(* IEC 61131-3 sources: std_i2980_v2.06_cp053/Source/IMM/ieccontrol/GlobalBaseArchives (part 10) *)

(* ---- ABLintabLoader.pu ---- *)
(*
@h    ! WARNING !
@h    The Kemro K2 system (including software) only meets category B according to EN 954-1,
@h    thus it is not intended for usage in safety-relevant control applications in the field
@h    of personal safety (e.g. emergency stop).
@h    To implement potentially necessary safety-relevant control tasks, always use additional
@h    external safety devices that are intended for the particular purpose, and meet the necessary
@h    functional safety.
@h    For further information see EN 954-1 (EN ISO 13849-1) and/or the K2-x00 user manual, chapter
@h    "CE conformity, directives and standards".

lintab loader

@FunctionID: CR_0030048

*)

IMPORT_OVER_LISTFILE
 GET_RUNTIME
, KFILE_Open
, KFILE_Read
, KFILE_Close
, STRING_TO_ASCII
, KFILE_GetFirst
, KFILE_GetNext
, KCAT_GetHandle
, KCAT_GetValue
, CMD_LINTABLOAD
, CMD_LINTABLISTFILES
, cLTBLDR_ERR_UNKNOWNCMD
, KFILE_Mode_ReadOnly
, KFILE_Status_OK
, cLTBLDR_ERR_FILENOTFOUND
, cLTBLDR_ERR_OUTOFBOUND
, cLTBLDR_MAXFILES
, cLTBLDR_ERR_MAXFILESREACHED
, KCAT_Status_OK
, cLTBLDR_ROOTPATH
, tsLintabLoaderData
, KFILE_Status
, tsTraceLevel
, KFILE_Open_Data
, KCTRL_Lintab_Point
, KAPPL_LintabData
, KCAT_Status
, KCAT_HandleData

END_IMPORT

ALGORITHM_BLOCK ABLintabLoader #DUMMY_EDIT_BLOCK

SYSTEM_VAR
 sv_LintabLoaderData : tsLintabLoaderData;
 sv_TraceLevel : tsTraceLevel;
END_VAR

SYSTEM_OBJECT
 TaskVis : TASK;
 PU_Task_7 : TASK;
END_OBJECT

VAR
 mbCmdActive : BOOL;
 Status : KFILE_Status;
 absoluteLTBPath : STRING(255);
END_VAR

POSTUPDATE_ALGORITHM pRunHMICmd ON PU_Task_7 WITH sv_LintabLoaderData.HMIComm.iCmdCtrl

#BEGIN_EDIT_BLOCK
(**************************************** WARNING ********************************************
 *** The KEBA Kemro K2 System including software is not intended for safety control tasks! ***
 ***                       For further information see Comment tab!                        ***
 *********************************************************************************************)

IF ((sv_LintabLoaderData.HMIComm.iCmdCtrl MOD 2) = 1) THEN // start command req.
    IF mbCmdActive THEN
        RETURN;
    END_IF;

    CASE sv_LintabLoaderData.HMIComm.iCmdSel OF
        CMD_LINTABLOAD:
            mbCmdActive := TRUE;
            START_PROCESS_ALGORITHM(paLoad);

        CMD_LINTABLISTFILES:
            mbCmdActive := TRUE;
            START_PROCESS_ALGORITHM(paListFiles);
    ELSE
        sv_LintabLoaderData.HMIComm.iCmdRet := cLTBLDR_ERR_UNKNOWNCMD;
        sv_LintabLoaderData.HMIComm.iCmdCtrl := sv_LintabLoaderData.HMIComm.iCmdCtrl + 1;
    END_CASE;
END_IF;

;#END_EDIT_BLOCK END_ALGORITHM

ALGORITHM aCmdDone

VAR_INPUT
 iRetCode : DINT;
END_VAR

VAR
 iTmp : DINT;
END_VAR
#BEGIN_EDIT_BLOCK
(**************************************** WARNING ********************************************
 *** The KEBA Kemro K2 System including software is not intended for safety control tasks! ***
 ***                       For further information see Comment tab!                        ***
 *********************************************************************************************)

iTmp := sv_LintabLoaderData.HMIComm.iCmdCtrl;
iTmp := iTmp + (iTmp MOD 2);
sv_LintabLoaderData.HMIComm.iCmdCtrl := iTmp;  // i MOD 2 = 0
sv_LintabLoaderData.HMIComm.iCmdRet := iRetCode;
mbCmdActive := FALSE;

;#END_EDIT_BLOCK END_ALGORITHM

PROCESS_ALGORITHM paLoad ON TaskVis

VAR
 dummy : DINT;
 t : TIME;
 tl : DINT;
 i : DINT;
 iLine : DINT;
 FileOpenData : KFILE_Open_Data;
 sColumn : STRING(255);
 sChar : STRING(1);
 bConvert : BOOL;
 iColumn : DINT;
 tmpPoint : KCTRL_Lintab_Point;
 tmpLintab : KAPPL_LintabData (* do not make VAR_TEMP, workaround CR_36866 *);
 iMaxPoints : DINT;
 bNoData : BOOL;
 AsciiChar : BYTE;
 // testSX : STRING(255);
 // testSY : STRING(255);
 // testS : STRING(255);
END_VAR
#BEGIN_EDIT_BLOCK
(**************************************** WARNING ********************************************
 *** The KEBA Kemro K2 System including software is not intended for safety control tasks! ***
 ***                       For further information see Comment tab!                        ***
 *********************************************************************************************)

IF sv_TraceLevel.bApplication THEN
   dummy := Print ('LOAD %s', sv_LintabLoaderData.sName);
   t := GET_RUNTIME();
END_IF;

iLine := 0;
iColumn := 0;
sColumn := '';
bConvert := FALSE;
iMaxPoints := GET_HIGH_BOUND(tmpLintab.LintabPoints.Point);

FileOpenData := KFILE_Open(CONCAT(absoluteLTBPath, '/', sv_LintabLoaderData.sName, '/', sv_LintabLoaderData.HMIComm.sFileName), KFILE_Mode_ReadOnly);

IF FileOpenData.Status <> KFILE_Status_OK THEN
    aCmdDone(cLTBLDR_ERR_FILENOTFOUND);
    STOP_PROCESS_ALGORITHM();
    RETURN;
END_IF;

REPEAT
      // read character
      i := KFILE_Read(FileOpenData.Token, 1, sChar);

      // new line detected
      IF (sChar = '$R') OR (sChar = '$L') THEN
          iColumn := 0;
          bConvert := TRUE;
      END_IF;

      // new column detected
      IF (sChar = ';') THEN
          iColumn := 1;
          bConvert := TRUE;
      END_IF;

      // no more characters left
      IF (i = 0) THEN
          iColumn := iColumn + 1;
          bConvert := TRUE;
      END_IF;

      IF bConvert THEN
             // try to convert linedata to lintabdata if there were no invalid chars in line and length > 0
             IF (NOT bNoData) AND (LEN(sColumn) > 0) THEN
                  IF ((iColumn MOD 2) = 1) THEN
                     tmpPoint.rX := STRING_TO_REAL(sColumn);
                  ELSE
                     tmpPoint.rY := STRING_TO_REAL(sColumn);

                     // check array limits
                     IF iLine >= iMaxPoints THEN
                            tmpLintab.LintabPoints.uNoOfPoints := DINT_TO_UDINT(iLine);
                            sv_LintabLoaderData.pLintab^ := tmpLintab;
                            sv_LintabLoaderData.HMIComm.sActFileName := sv_LintabLoaderData.HMIComm.sFileName;
                            Status := KFILE_Close(FileOpenData.Token);
                            aCmdDone(cLTBLDR_ERR_OUTOFBOUND);
                            STOP_PROCESS_ALGORITHM();
                            RETURN;
                     END_IF;

                     iLine := iLine + 1;
                     tmpLintab.LintabPoints.Point[iLine] := tmpPoint;
                  END_IF;
             END_IF;
             IF (iColumn MOD 2) = 0 THEN // if x value invalid, do not try to convert y; so only reset bNoData if y value reached
                 bNoData := FALSE;
             END_IF;
             sColumn := '';
             bConvert := FALSE;
      END_IF;
      IF i = 1 THEN
         AsciiChar:=STRING_TO_ASCII(sChar);
         IF (NOT bNoData) AND (AsciiChar > 16#20) AND (sChar <> ';') THEN // ignore control chars (ascii code 0x20 and lower), ignore if there where invalid chars previously, ignore column seperator
                 IF ((AsciiChar >= 16#30) AND (AsciiChar < 16#40)) // digit
                     OR (sChar = '.') OR (sChar = '-') OR (sChar = '+') THEN
                   sColumn := CONCAT(sColumn, sChar);
                 ELSE
                   bNoData := TRUE; // invalid char detected
                 END_IF;
         END_IF;
      END_IF;
UNTIL i = 0
END_REPEAT;

Status := KFILE_Close(FileOpenData.Token);

IF sv_TraceLevel.bApplication THEN
   tl := LINT_TO_DINT(TIME_TO_LINT((GET_RUNTIME() - t)/1000));
   dummy := Print ('LOAD done %s; time: %d ms', sv_LintabLoaderData.sName, tl);
END_IF;

tmpLintab.LintabPoints.uNoOfPoints := DINT_TO_UDINT(iLine);
sv_LintabLoaderData.pLintab^ := tmpLintab;
sv_LintabLoaderData.HMIComm.sActFileName := sv_LintabLoaderData.HMIComm.sFileName;
aCmdDone(0);
STOP_PROCESS_ALGORITHM();

//debug
(*FOR i:=1 TO iLine DO
    tmpPoint := tmpLintab.LintabPoints.Point[i];
    testSX := REAL_TO_FORMATTED_STRING(tmpPoint.rX, 10, 5);
    testSY := REAL_TO_FORMATTED_STRING(tmpPoint.rY,10, 5);
    testS := CONCAT(testSX, ';', testSY);
    dummy:=Print("%s", testS);
END_FOR;
*)

;#END_EDIT_BLOCK END_ALGORITHM

PROCESS_ALGORITHM paListFiles ON TaskVis

VAR
 dummy : DINT;
 sFile : STRING(255);
 i : DINT;
 t : TIME;
 tl : DINT;
 iLenRootPath : DINT;
END_VAR
#BEGIN_EDIT_BLOCK
(**************************************** WARNING ********************************************
 *** The KEBA Kemro K2 System including software is not intended for safety control tasks! ***
 ***                       For further information see Comment tab!                        ***
 *********************************************************************************************)

IF sv_TraceLevel.bApplication THEN
   dummy := Print ('LIST %s', sv_LintabLoaderData.sName);
   t := GET_RUNTIME();
END_IF;

i := 0;
Status := KFILE_GetFirst(CONCAT(absoluteLTBPath, '/', sv_LintabLoaderData.sName), sFile);
iLenRootPath := LEN(CONCAT(absoluteLTBPath, '/', sv_LintabLoaderData.sName, '/'));

WHILE (Status = KFILE_Status_OK) DO
    i := i + 1;
    IF i > cLTBLDR_MAXFILES THEN

        IF sv_TraceLevel.bApplication THEN
           tl := LINT_TO_DINT(TIME_TO_LINT((GET_RUNTIME() - t)/1000));
           dummy := Print ('LIST Done %s; time: %d ms', sv_LintabLoaderData.sName, tl);
        END_IF;

        sv_LintabLoaderData.HMIComm.FileList.iFileCount := cLTBLDR_MAXFILES;
        aCmdDone(cLTBLDR_ERR_MAXFILESREACHED);
        STOP_PROCESS_ALGORITHM();
        RETURN;
    END_IF;
    sv_LintabLoaderData.HMIComm.FileList.yFile[i] := RIGHT(sFile, LEN(sFile) - iLenRootPath);
    Status := KFILE_GetNext(sFile, sFile);
END_WHILE;

IF sv_TraceLevel.bApplication THEN
   tl := LINT_TO_DINT(TIME_TO_LINT((GET_RUNTIME() - t)/1000));
   dummy := Print ('LIST Done %s; time: %d ms', sv_LintabLoaderData.sName, tl);
END_IF;

sv_LintabLoaderData.HMIComm.FileList.iFileCount := i;
aCmdDone(0);
STOP_PROCESS_ALGORITHM();

;#END_EDIT_BLOCK END_ALGORITHM

PROCESS_ALGORITHM paInit ON TaskVis AUTOSTART

VAR
 Status_CAT : KCAT_Status;
 StatusName_CAT : KCAT_HandleData;
 sRootPath : STRING(255);
END_VAR
#BEGIN_EDIT_BLOCK
(**************************************** WARNING ********************************************
 *** The KEBA Kemro K2 System including software is not intended for safety control tasks! ***
 ***                       For further information see Comment tab!                        ***
 *********************************************************************************************)

StatusName_CAT := KCAT_GetHandle('System.workPath');
IF StatusName_CAT.Status = KCAT_Status_OK THEN
    Status_CAT := KCAT_GetValue(Handle := StatusName_CAT.Handle, Buffer := sRootPath);
END_IF;

absoluteLTBPath := CONCAT(sRootPath,cLTBLDR_ROOTPATH);
STOP_PROCESS_ALGORITHM();

;#END_EDIT_BLOCK END_ALGORITHM

END_ALGORITHM_BLOCK

#END_OF_IEC_PART

@Puma @IecEditor 6 103 @Pou 25
@@@BEG_Comment@@@
@h    ! WARNING !
@h    The Kemro K2 system (including software) only meets category B according to EN 954-1,
@h    thus it is not intended for usage in safety-relevant control applications in the field
@h    of personal safety (e.g. emergency stop).
@h    To implement potentially necessary safety-relevant control tasks, always use additional
@h    external safety devices that are intended for the particular purpose, and meet the necessary
@h    functional safety.
@h    For further information see EN 954-1 (EN ISO 13849-1) and/or the K2-x00 user manual, chapter
@h    "CE conformity, directives and standards".

lintab loader

@FunctionID: CR_0030048

@@@END_Comment@@@

@BEG_Contents

@BEG_Func
@RT(17)FuncTreeContainer
9
@Var @RT(11)GET_RUNTIME @RT(0) @T @T @DERIVED 0 @F @RT(22)KEBA_STANDARD_FUNCTION @F
@T
@BEG_Attrib
0 @RT(0) @RT(0)
@END_Attrib
1 1 @F @F @F @F

@Var @RT(10)KFILE_Open @RT(0) @T @T @DERIVED 0 @F @RT(22)KEBA_STANDARD_FUNCTION @F
@T
@BEG_Attrib
0 @RT(0) @RT(0)
@END_Attrib
1 1 @F @F @F @F

@Var @RT(10)KFILE_Read @RT(0) @T @T @DERIVED 0 @F @RT(22)KEBA_STANDARD_FUNCTION @F
@T
@BEG_Attrib
0 @RT(0) @RT(0)
@END_Attrib
1 1 @F @F @F @F

@Var @RT(11)KFILE_Close @RT(0) @T @T @DERIVED 0 @F @RT(22)KEBA_STANDARD_FUNCTION @F
@T
@BEG_Attrib
0 @RT(0) @RT(0)
@END_Attrib
1 1 @F @F @F @F

@Var @RT(15)STRING_TO_ASCII @RT(0) @T @T @DERIVED 0 @F @RT(22)KEBA_STANDARD_FUNCTION @F
@T
@BEG_Attrib
0 @RT(0) @RT(0)
@END_Attrib
1 1 @F @F @F @F

@Var @RT(14)KFILE_GetFirst @RT(0) @T @T @DERIVED 0 @F @RT(22)KEBA_STANDARD_FUNCTION @F
@T
@BEG_Attrib
0 @RT(0) @RT(0)
@END_Attrib
1 1 @F @F @F @F

@Var @RT(13)KFILE_GetNext @RT(0) @T @T @DERIVED 0 @F @RT(22)KEBA_STANDARD_FUNCTION @F
@T
@BEG_Attrib
0 @RT(0) @RT(0)
@END_Attrib
1 1 @F @F @F @F

@Var @RT(14)KCAT_GetHandle @RT(0) @T @T @DERIVED 0 @F @RT(22)KEBA_STANDARD_FUNCTION @F
@T
@BEG_Attrib
0 @RT(0) @RT(0)
@END_Attrib
1 1 @F @F @F @F

@Var @RT(13)KCAT_GetValue @RT(0) @T @T @DERIVED 0 @F @RT(22)KEBA_STANDARD_FUNCTION @F
@T
@BEG_Attrib
0 @RT(0) @RT(0)
@END_Attrib
1 1 @F @F @F @F

@END_Func

@BEG_Const
@RT(18)ConstTreeContainer
11
@Var @RT(14)CMD_LINTABLOAD @RT(0) @T @F @DT @RT(4)DINT @RT(0) @T @T @BASIC 0 @F
@F @F
@T
@BEG_Attrib
0 @RT(1)0 @RT(0)
@END_Attrib
1 1 @F @F @F @F

@Var @RT(19)CMD_LINTABLISTFILES @RT(0) @T @F @DT @RT(4)DINT @RT(0) @T @T @BASIC 0 @F
@F @F
@T
@BEG_Attrib
0 @RT(1)1 @RT(0)
@END_Attrib
1 1 @F @F @F @F

@Var @RT(22)cLTBLDR_ERR_UNKNOWNCMD @RT(0) @T @F @DT @RT(4)DINT @RT(0) @T @T @BASIC 0 @F
@F @F
@T
@BEG_Attrib
0 @RT(1)1 @RT(0)
@END_Attrib
1 1 @F @F @F @F

@Var @RT(19)KFILE_Mode_ReadOnly @RT(0) @T @T @DERIVED 0 @F @RT(10)KFILE_Mode @F
@T
@BEG_Attrib
0 @RT(1)0 @RT(22)opens for reading only
@END_Attrib
1 1 @F @F @F @F

@Var @RT(15)KFILE_Status_OK @RT(0) @T @T @DERIVED 0 @F @RT(12)KFILE_Status @F
@T
@BEG_Attrib
0 @RT(1)1 @RT(18)command successful
@END_Attrib
1 1 @F @F @F @F

@Var @RT(24)cLTBLDR_ERR_FILENOTFOUND @RT(0) @T @F @DT @RT(4)DINT @RT(0) @T @T @BASIC 0 @F
@F @F
@T
@BEG_Attrib
0 @RT(12)16#0002_0001 @RT(0)
@END_Attrib
1 1 @F @F @F @F

@Var @RT(22)cLTBLDR_ERR_OUTOFBOUND @RT(0) @T @F @DT @RT(4)DINT @RT(0) @T @T @BASIC 0 @F
@F @F
@T
@BEG_Attrib
0 @RT(12)16#0002_0002 @RT(0)
@END_Attrib
1 1 @F @F @F @F

@Var @RT(16)cLTBLDR_MAXFILES @RT(0) @T @F @DT @RT(4)DINT @RT(0) @T @T @BASIC 0 @F
@F @F
@T
@BEG_Attrib
0 @RT(2)20 @RT(0)
@END_Attrib
1 1 @F @F @F @F

@Var @RT(27)cLTBLDR_ERR_MAXFILESREACHED @RT(0) @T @F @DT @RT(4)DINT @RT(0) @T @T @BASIC 0 @F
@F @F
@T
@BEG_Attrib
0 @RT(12)16#0001_0001 @RT(0)
@END_Attrib
1 1 @F @F @F @F

@Var @RT(14)KCAT_Status_OK @RT(0) @T @T @DERIVED 0 @F @RT(11)KCAT_Status @F
@T
@BEG_Attrib
0 @RT(1)0 @RT(0)
@END_Attrib
1 1 @F @F @F @F

@Var @RT(16)cLTBLDR_ROOTPATH @RT(0) @T @F @DT @RT(11)STRING(255) @RT(0) @T @T @STRING 0 @F @RT(3)255 @F
@F @F
@T
@BEG_Attrib
0 @RT(25)'/workspace/data/lintab/' @RT(0)
@END_Attrib
1 1 @F @F @F @F

@END_Const

@BEG_Export

@BEG_Kind
@ALGORITHM_BLOCK @RT(14)ABLintabLoader @STRUCTURED_TEXT
@RT(0) @RT(0) @RT(0)
@END_Kind

@BEG_Dcl
@RT(16)DclTreeContainer
7
@Var @RT(19)sv_LintabLoaderData @RT(0) @T @T @DERIVED 0 @T @T @DT @RT(18)tsLintabLoaderData @RT(0) @T @T @UNKNOWN 0 @F
@F @F
@T
@BEG_Attrib
3 @RT(0) @RT(0) @RT(0)
@END_Attrib
1 8 @F @F @F @F

@Var @RT(7)TaskVis @RT(0) @T @F @DT @RT(4)TASK @RT(0) @T @T @BASIC 0 @F
@F @F
@T
@BEG_Attrib
3 @RT(0) @RT(0) @RT(0)
@END_Attrib
1 7 @F @F @F @F

@Var @RT(9)PU_Task_7 @RT(0) @T @F @DT @RT(4)TASK @RT(0) @T @T @BASIC 0 @F
@F @F
@T
@BEG_Attrib
3 @RT(0) @RT(0) @RT(0)
@END_Attrib
1 7 @F @F @F @F

@Var @RT(11)mbCmdActive @RT(0) @T @F @DT @RT(4)BOOL @RT(0) @T @T @BASIC 0 @F
@F @F
@T
@BEG_Attrib
3 @RT(0) @RT(0) @RT(0)
@END_Attrib
1 0 @F @F @F @F

@Var @RT(6)Status @RT(0) @T @T @DERIVED 0 @T @T @DT @RT(12)KFILE_Status @RT(0) @T @T @UNKNOWN 0 @F
@F @F
@T
@BEG_Attrib
3 @RT(0) @RT(0) @RT(0)
@END_Attrib
1 0 @F @F @F @F

@Var @RT(15)absoluteLTBPath @RT(0) @T @F @DT @RT(11)STRING(255) @RT(0) @T @T @STRING 0 @F @RT(3)255 @F
@F @F
@T
@BEG_Attrib
3 @RT(0) @RT(0) @RT(0)
@END_Attrib
1 0 @F @F @F @F

@Var @RT(13)sv_TraceLevel @RT(0) @T @T @DERIVED 0 @F @RT(12)tsTraceLevel @F
@T
@BEG_Attrib
3 @RT(0) @RT(0) @RT(0)
@END_Attrib
1 8 @F @F @F @F

@END_Dcl

@END_Export

@BEG_Body

5

@BEG_Export

@BEG_Algo
@POSTUPDATE_ALGORITHM @RT(10)pRunHMICmd @STRUCTURED_TEXT
@RT(0) @RT(36)sv_LintabLoaderData.HMIComm.iCmdCtrl @RT(9)PU_Task_7 @F @F
@END_Algo

@BEG_Dcl
@RT(16)DclTreeContainer
0
@END_Dcl

@END_Export

@BEG_Export

@BEG_Algo
@ALGORITHM @RT(8)aCmdDone @STRUCTURED_TEXT
@RT(0) @RT(0) @RT(0) @F @F
@END_Algo

@BEG_Dcl
@RT(16)DclTreeContainer
2
@Var @RT(8)iRetCode @RT(0) @T @F @DT @RT(4)DINT @RT(0) @T @T @BASIC 0 @F
@F @F
@T
@BEG_Attrib
3 @RT(0) @RT(0) @RT(0)
@END_Attrib
1 1 @F @F @F @F

@Var @RT(4)iTmp @RT(0) @T @F @DT @RT(4)DINT @RT(0) @T @T @BASIC 0 @F
@F @F
@T
@BEG_Attrib
3 @RT(0) @RT(0) @RT(0)
@END_Attrib
1 0 @F @F @F @F

@END_Dcl

@END_Export

@BEG_Export

@BEG_Algo
@PROCESS_ALGORITHM @RT(6)paLoad @STRUCTURED_TEXT
@RT(0) @RT(0) @RT(7)TaskVis @F @F
@END_Algo

@BEG_Dcl
@RT(16)DclTreeContainer
18
@Var @RT(5)dummy @RT(0) @T @F @DT @RT(4)DINT @RT(0) @T @T @BASIC 0 @F
@F @F
@T
@BEG_Attrib
3 @RT(0) @RT(0) @RT(0)
@END_Attrib
1 0 @F @F @F @F

@Var @RT(1)t @RT(0) @T @F @DT @RT(4)TIME @RT(0) @T @T @BASIC 0 @F
@F @F
@T
@BEG_Attrib
3 @RT(0) @RT(0) @RT(0)
@END_Attrib
1 0 @F @F @F @F

@Var @RT(2)tl @RT(0) @T @F @DT @RT(4)DINT @RT(0) @T @T @BASIC 0 @F
@F @F
@T
@BEG_Attrib
3 @RT(0) @RT(0) @RT(0)
@END_Attrib
1 0 @F @F @F @F

@Var @RT(1)i @RT(0) @T @F @DT @RT(4)DINT @RT(0) @T @T @BASIC 0 @F
@F @F
@T
@BEG_Attrib
3 @RT(0) @RT(0) @RT(0)
@END_Attrib
1 0 @F @F @F @F

@Var @RT(5)iLine @RT(0) @T @F @DT @RT(4)DINT @RT(0) @T @T @BASIC 0 @F
@F @F
@T
@BEG_Attrib
3 @RT(0) @RT(0) @RT(0)
@END_Attrib
1 0 @F @F @F @F

@Var @RT(12)FileOpenData @RT(0) @T @T @DERIVED 0 @T @T @DT @RT(15)KFILE_Open_Data @RT(0) @T @T @UNKNOWN 0 @F
@F @F
@T
@BEG_Attrib
3 @RT(0) @RT(0) @RT(0)
@END_Attrib
1 0 @F @F @F @F

@Var @RT(7)sColumn @RT(0) @T @F @DT @RT(11)STRING(255) @RT(0) @T @T @STRING 0 @F @RT(3)255 @F
@F @F
@T
@BEG_Attrib
3 @RT(0) @RT(0) @RT(0)
@END_Attrib
1 0 @F @F @F @F

@Var @RT(5)sChar @RT(0) @T @F @DT @RT(9)STRING(1) @RT(0) @T @T @STRING 0 @F @RT(1)1 @F
@F @F
@T
@BEG_Attrib
3 @RT(0) @RT(0) @RT(0)
@END_Attrib
1 0 @F @F @F @F

@Var @RT(8)bConvert @RT(0) @T @F @DT @RT(4)BOOL @RT(0) @T @T @BASIC 0 @F
@F @F
@T
@BEG_Attrib
3 @RT(0) @RT(0) @RT(0)
@END_Attrib
1 0 @F @F @F @F

@Var @RT(7)iColumn @RT(0) @T @F @DT @RT(4)DINT @RT(0) @T @T @BASIC 0 @F
@F @F
@T
@BEG_Attrib
3 @RT(0) @RT(0) @RT(0)
@END_Attrib
1 0 @F @F @F @F

@Var @RT(8)tmpPoint @RT(0) @T @T @DERIVED 0 @T @T @DT @RT(18)KCTRL_Lintab_Point @RT(0) @T @T @UNKNOWN 0 @F
@F @F
@T
@BEG_Attrib
3 @RT(0) @RT(0) @RT(0)
@END_Attrib
1 0 @F @F @F @F

@Var @RT(9)tmpLintab @RT(0) @T @T @DERIVED 0 @T @T @DT @RT(16)KAPPL_LintabData @RT(0) @T @T @UNKNOWN 0 @F
@F @F
@T
@BEG_Attrib
3 @RT(0) @RT(41)do not make VAR_TEMP, workaround CR_36866 @RT(0)
@END_Attrib
1 0 @F @F @F @F

@Var @RT(10)iMaxPoints @RT(0) @T @F @DT @RT(4)DINT @RT(0) @T @T @BASIC 0 @F
@F @F
@T
@BEG_Attrib
3 @RT(0) @RT(0) @RT(0)
@END_Attrib
1 0 @F @F @F @F

@Var @RT(7)bNoData @RT(0) @T @F @DT @RT(4)BOOL @RT(0) @T @T @BASIC 0 @F
@F @F
@T
@BEG_Attrib
3 @RT(0) @RT(0) @RT(0)
@END_Attrib
1 0 @F @F @F @F

@Var @RT(9)AsciiChar @RT(0) @T @F @DT @RT(4)BYTE @RT(0) @T @T @BASIC 0 @F
@F @F
@T
@BEG_Attrib
3 @RT(0) @RT(0) @RT(0)
@END_Attrib
1 0 @F @F @F @F

@Var @RT(6)testSX @RT(0) @T @F @DT @RT(11)STRING(255) @RT(0) @T @T @STRING 0 @F @RT(3)255 @F
@F @T
@T
@BEG_Attrib
3 @RT(0) @RT(0) @RT(0)
@END_Attrib
1 0 @F @F @F @F

@Var @RT(6)testSY @RT(0) @T @F @DT @RT(11)STRING(255) @RT(0) @T @T @STRING 0 @F @RT(3)255 @F
@F @T
@T
@BEG_Attrib
3 @RT(0) @RT(0) @RT(0)
@END_Attrib
1 0 @F @F @F @F

@Var @RT(5)testS @RT(0) @T @F @DT @RT(11)STRING(255) @RT(0) @T @T @STRING 0 @F @RT(3)255 @F
@F @T
@T
@BEG_Attrib
3 @RT(0) @RT(0) @RT(0)
@END_Attrib
1 0 @F @F @F @F

@END_Dcl

@END_Export

@BEG_Export

@BEG_Algo
@PROCESS_ALGORITHM @RT(11)paListFiles @STRUCTURED_TEXT
@RT(0) @RT(0) @RT(7)TaskVis @F @F
@END_Algo

@BEG_Dcl
@RT(16)DclTreeContainer
6
@Var @RT(5)dummy @RT(0) @T @F @DT @RT(4)DINT @RT(0) @T @T @BASIC 0 @F
@F @F
@T
@BEG_Attrib
3 @RT(0) @RT(0) @RT(0)
@END_Attrib
1 0 @F @F @F @F

@Var @RT(5)sFile @RT(0) @T @F @DT @RT(11)STRING(255) @RT(0) @T @T @STRING 0 @F @RT(3)255 @F
@F @F
@T
@BEG_Attrib
3 @RT(0) @RT(0) @RT(0)
@END_Attrib
1 0 @F @F @F @F

@Var @RT(1)i @RT(0) @T @F @DT @RT(4)DINT @RT(0) @T @T @BASIC 0 @F
@F @F
@T
@BEG_Attrib
3 @RT(0) @RT(0) @RT(0)
@END_Attrib
1 0 @F @F @F @F

@Var @RT(1)t @RT(0) @T @F @DT @RT(4)TIME @RT(0) @T @T @BASIC 0 @F
@F @F
@T
@BEG_Attrib
3 @RT(0) @RT(0) @RT(0)
@END_Attrib
1 0 @F @F @F @F

@Var @RT(2)tl @RT(0) @T @F @DT @RT(4)DINT @RT(0) @T @T @BASIC 0 @F
@F @F
@T
@BEG_Attrib
3 @RT(0) @RT(0) @RT(0)
@END_Attrib
1 0 @F @F @F @F

@Var @RT(12)iLenRootPath @RT(0) @T @F @DT @RT(4)DINT @RT(0) @T @T @BASIC 0 @F
@F @F
@T
@BEG_Attrib
3 @RT(0) @RT(0) @RT(0)
@END_Attrib
1 0 @F @F @F @F

@END_Dcl

@END_Export

@BEG_Export

@BEG_Algo
@PROCESS_ALGORITHM @RT(6)paInit @STRUCTURED_TEXT
@RT(0) @RT(0) @RT(7)TaskVis @T @F
@END_Algo

@BEG_Dcl
@RT(16)DclTreeContainer
3
@Var @RT(10)Status_CAT @RT(0) @T @T @DERIVED 0 @T @T @DT @RT(11)KCAT_Status @RT(0) @T @T @UNKNOWN 0 @F
@F @F
@T
@BEG_Attrib
3 @RT(0) @RT(0) @RT(0)
@END_Attrib
1 0 @F @F @F @F

@Var @RT(14)StatusName_CAT @RT(0) @T @T @DERIVED 0 @T @T @DT @RT(15)KCAT_HandleData @RT(0) @T @T @UNKNOWN 0 @F
@F @F
@T
@BEG_Attrib
3 @RT(0) @RT(0) @RT(0)
@END_Attrib
1 0 @F @F @F @F

@Var @RT(9)sRootPath @RT(0) @T @F @DT @RT(11)STRING(255) @RT(0) @T @T @STRING 0 @F @RT(3)255 @F
@F @F
@T
@BEG_Attrib
3 @RT(0) @RT(0) @RT(0)
@END_Attrib
1 0 @F @F @F @F

@END_Dcl

@END_Export

@BEG_Body
@TL(24)
(**************************************** WARNING ********************************************
 *** The KEBA Kemro K2 System including software is not intended for safety control tasks! ***
 ***                       For further information see Comment tab!                        ***
 *********************************************************************************************)

IF ((sv_LintabLoaderData.HMIComm.iCmdCtrl MOD 2) = 1) THEN // start command req.
    IF mbCmdActive THEN
        RETURN;
    END_IF;

    CASE sv_LintabLoaderData.HMIComm.iCmdSel OF
        CMD_LINTABLOAD:
            mbCmdActive := TRUE;
            START_PROCESS_ALGORITHM(paLoad);

        CMD_LINTABLISTFILES:
            mbCmdActive := TRUE;
            START_PROCESS_ALGORITHM(paListFiles);
    ELSE
        sv_LintabLoaderData.HMIComm.iCmdRet := cLTBLDR_ERR_UNKNOWNCMD;
        sv_LintabLoaderData.HMIComm.iCmdCtrl := sv_LintabLoaderData.HMIComm.iCmdCtrl + 1;
    END_CASE;
END_IF;

@END_Body

@@@BEG_Comment@@@
@TL(0)

@@@END_Comment@@@

@BEG_Body
@TL(12)
(**************************************** WARNING ********************************************
 *** The KEBA Kemro K2 System including software is not intended for safety control tasks! ***
 ***                       For further information see Comment tab!                        ***
 *********************************************************************************************)

iTmp := sv_LintabLoaderData.HMIComm.iCmdCtrl;
iTmp := iTmp + (iTmp MOD 2);
sv_LintabLoaderData.HMIComm.iCmdCtrl := iTmp;  // i MOD 2 = 0
sv_LintabLoaderData.HMIComm.iCmdRet := iRetCode;
mbCmdActive := FALSE;

@END_Body

@@@BEG_Comment@@@
@TL(0)

@@@END_Comment@@@

@BEG_Body
@TL(112)
(**************************************** WARNING ********************************************
 *** The KEBA Kemro K2 System including software is not intended for safety control tasks! ***
 ***                       For further information see Comment tab!                        ***
 *********************************************************************************************)

IF sv_TraceLevel.bApplication THEN
   dummy := Print ('LOAD %s', sv_LintabLoaderData.sName);
   t := GET_RUNTIME();
END_IF;

iLine := 0;
iColumn := 0;
sColumn := '';
bConvert := FALSE;
iMaxPoints := GET_HIGH_BOUND(tmpLintab.LintabPoints.Point);

FileOpenData := KFILE_Open(CONCAT(absoluteLTBPath, '/', sv_LintabLoaderData.sName, '/', sv_LintabLoaderData.HMIComm.sFileName), KFILE_Mode_ReadOnly);

IF FileOpenData.Status <> KFILE_Status_OK THEN
    aCmdDone(cLTBLDR_ERR_FILENOTFOUND);
    STOP_PROCESS_ALGORITHM();
    RETURN;
END_IF;

REPEAT
      // read character
      i := KFILE_Read(FileOpenData.Token, 1, sChar);

      // new line detected
      IF (sChar = '$R') OR (sChar = '$L') THEN
          iColumn := 0;
          bConvert := TRUE;
      END_IF;

      // new column detected
      IF (sChar = ';') THEN
          iColumn := 1;
          bConvert := TRUE;
      END_IF;

      // no more characters left
      IF (i = 0) THEN
          iColumn := iColumn + 1;
          bConvert := TRUE;
      END_IF;

      IF bConvert THEN
             // try to convert linedata to lintabdata if there were no invalid chars in line and length > 0
             IF (NOT bNoData) AND (LEN(sColumn) > 0) THEN
                  IF ((iColumn MOD 2) = 1) THEN
                     tmpPoint.rX := STRING_TO_REAL(sColumn);
                  ELSE
                     tmpPoint.rY := STRING_TO_REAL(sColumn);

                     // check array limits
                     IF iLine >= iMaxPoints THEN
                            tmpLintab.LintabPoints.uNoOfPoints := DINT_TO_UDINT(iLine);
                            sv_LintabLoaderData.pLintab^ := tmpLintab;
                            sv_LintabLoaderData.HMIComm.sActFileName := sv_LintabLoaderData.HMIComm.sFileName;
                            Status := KFILE_Close(FileOpenData.Token);
                            aCmdDone(cLTBLDR_ERR_OUTOFBOUND);
                            STOP_PROCESS_ALGORITHM();
                            RETURN;
                     END_IF;

                     iLine := iLine + 1;
                     tmpLintab.LintabPoints.Point[iLine] := tmpPoint;
                  END_IF;
             END_IF;
             IF (iColumn MOD 2) = 0 THEN // if x value invalid, do not try to convert y; so only reset bNoData if y value reached
                 bNoData := FALSE;
             END_IF;
             sColumn := '';
             bConvert := FALSE;
      END_IF;
      IF i = 1 THEN
         AsciiChar:=STRING_TO_ASCII(sChar);
         IF (NOT bNoData) AND (AsciiChar > 16#20) AND (sChar <> ';') THEN // ignore control chars (ascii code 0x20 and lower), ignore if there where invalid chars previously, ignore column seperator
                 IF ((AsciiChar >= 16#30) AND (AsciiChar < 16#40)) // digit
                     OR (sChar = '.') OR (sChar = '-') OR (sChar = '+') THEN
                   sColumn := CONCAT(sColumn, sChar);
                 ELSE
                   bNoData := TRUE; // invalid char detected
                 END_IF;
         END_IF;
      END_IF;
UNTIL i = 0
END_REPEAT;

Status := KFILE_Close(FileOpenData.Token);

IF sv_TraceLevel.bApplication THEN
   tl := LINT_TO_DINT(TIME_TO_LINT((GET_RUNTIME() - t)/1000));
   dummy := Print ('LOAD done %s; time: %d ms', sv_LintabLoaderData.sName, tl);
END_IF;

tmpLintab.LintabPoints.uNoOfPoints := DINT_TO_UDINT(iLine);
sv_LintabLoaderData.pLintab^ := tmpLintab;
sv_LintabLoaderData.HMIComm.sActFileName := sv_LintabLoaderData.HMIComm.sFileName;
aCmdDone(0);
STOP_PROCESS_ALGORITHM();

//debug
(*FOR i:=1 TO iLine DO
    tmpPoint := tmpLintab.LintabPoints.Point[i];
    testSX := REAL_TO_FORMATTED_STRING(tmpPoint.rX, 10, 5);
    testSY := REAL_TO_FORMATTED_STRING(tmpPoint.rY,10, 5);
    testS := CONCAT(testSX, ';', testSY);
    dummy:=Print("%s", testS);
END_FOR;
*)

@END_Body

@@@BEG_Comment@@@
@TL(0)

@@@END_Comment@@@

@BEG_Body
@TL(41)
(**************************************** WARNING ********************************************
 *** The KEBA Kemro K2 System including software is not intended for safety control tasks! ***
 ***                       For further information see Comment tab!                        ***
 *********************************************************************************************)

IF sv_TraceLevel.bApplication THEN
   dummy := Print ('LIST %s', sv_LintabLoaderData.sName);
   t := GET_RUNTIME();
END_IF;

i := 0;
Status := KFILE_GetFirst(CONCAT(absoluteLTBPath, '/', sv_LintabLoaderData.sName), sFile);
iLenRootPath := LEN(CONCAT(absoluteLTBPath, '/', sv_LintabLoaderData.sName, '/'));

WHILE (Status = KFILE_Status_OK) DO
    i := i + 1;
    IF i > cLTBLDR_MAXFILES THEN

        IF sv_TraceLevel.bApplication THEN
           tl := LINT_TO_DINT(TIME_TO_LINT((GET_RUNTIME() - t)/1000));
           dummy := Print ('LIST Done %s; time: %d ms', sv_LintabLoaderData.sName, tl);
        END_IF;

        sv_LintabLoaderData.HMIComm.FileList.iFileCount := cLTBLDR_MAXFILES;
        aCmdDone(cLTBLDR_ERR_MAXFILESREACHED);
        STOP_PROCESS_ALGORITHM();
        RETURN;
    END_IF;
    sv_LintabLoaderData.HMIComm.FileList.yFile[i] := RIGHT(sFile, LEN(sFile) - iLenRootPath);
    Status := KFILE_GetNext(sFile, sFile);
END_WHILE;

IF sv_TraceLevel.bApplication THEN
   tl := LINT_TO_DINT(TIME_TO_LINT((GET_RUNTIME() - t)/1000));
   dummy := Print ('LIST Done %s; time: %d ms', sv_LintabLoaderData.sName, tl);
END_IF;

sv_LintabLoaderData.HMIComm.FileList.iFileCount := i;
aCmdDone(0);
STOP_PROCESS_ALGORITHM();

@END_Body

@@@BEG_Comment@@@
@TL(0)

@@@END_Comment@@@

@BEG_Body
@TL(13)
(**************************************** WARNING ********************************************
 *** The KEBA Kemro K2 System including software is not intended for safety control tasks! ***
 ***                       For further information see Comment tab!                        ***
 *********************************************************************************************)

StatusName_CAT := KCAT_GetHandle('System.workPath');
IF StatusName_CAT.Status = KCAT_Status_OK THEN
    Status_CAT := KCAT_GetValue(Handle := StatusName_CAT.Handle, Buffer := sRootPath);
END_IF;

absoluteLTBPath := CONCAT(sRootPath,cLTBLDR_ROOTPATH);
STOP_PROCESS_ALGORITHM();

@END_Body

@@@BEG_Comment@@@
@TL(0)

@@@END_Comment@@@
@END_Body

@END_Contents

(* ---- ABList.pu ---- *)
(*
@h    ! WARNING !
@h    The Kemro K2 system (including software) only meets category B according to EN 954-1,
@h    thus it is not intended for usage in safety-relevant control applications in the field
@h    of personal safety (e.g. emergency stop).
@h    To implement potentially necessary safety-relevant control tasks, always use additional
@h    external safety devices that are intended for the particular purpose, and meet the necessary
@h    functional safety.
@h    For further information see EN 954-1 (EN ISO 13849-1) and/or the K2-x00 user manual, chapter
@h    "CE conformity, directives and standards".

This AB is a model of a list-administration. It provides methods for adding, removing, searching
and fetching listelements.
The list is seperated in 2 dataparts:
- mListStruct.List[x].SearchData
- mListStruct.List[x].ElementData
SearchData is the data which is used for searching an entry in the list.
ElementData is a additional datapart.

The block must be adapted before it is ready for use.
For customizing the list, new listtypes have to be created. (see the models in ListTypes.tu)
This can be done easily by replacing the string "XY" by any list identifier.
Example: To create a Motorlist copy and adapt the datatypes of ListTypes.tu.
          Search and replace "XY" by "Motor"  -> tsListStructMotor.
         Rename ABList.pu and Search and replace "XY" by "Motor".

*)

IMPORT_OVER_LISTFILE
 SET_ALARM
, tsListStructXY
, tsDeviceId
, FBDebugTrace
, tsTraceLevel
, tsElementXY
, tsSearchDataXY

END_IMPORT

ALGORITHM_BLOCK ABList #DUMMY_EDIT_BLOCK

SYSTEM_VAR
 sv_DeviceId : tsDeviceId;
 sv_TraceLevel : tsTraceLevel;
END_VAR

SYSTEM_OBJECT
 erListOverflow : ALARM;
END_OBJECT

VAR
 mListStruct : tsListStructXY;
 miNextFree : DINT;
 miLowBound : DINT;
 miHighBound : DINT;
 mbInit : BOOL;
 miLastFound : DINT;
 miActElement : DINT;
 fbDebugTrace : FBDebugTrace;
END_VAR

ALGORITHM aInit

#BEGIN_EDIT_BLOCK
miLowBound := GET_LOW_BOUND(mListStruct.List);
miHighBound := GET_HIGH_BOUND(mListStruct.List);
miNextFree := miLowBound;
miLastFound := miLowBound;
miActElement := miLowBound;
mbInit := TRUE;

;#END_EDIT_BLOCK END_ALGORITHM

ALGORITHM aAdd

VAR_INPUT
 Element : tsElementXY;
END_VAR
#BEGIN_EDIT_BLOCK
IF NOT mbInit THEN RETURN;; END_IF;

IF miNextFree < miHighBound THEN

    mListStruct.List[miNextFree] := Element;
    mListStruct.Used[miNextFree] := TRUE;
    miNextFree := miNextFree + 1;
ELSE
    //error: List Full
    SET_ALARM(Name := erListOverflow,
              SubID1 := sv_DeviceId.CompId,
              SubID2 := sv_DeviceId.IndexId,
              Param1 := 'ABList.aAdd');
END_IF;

;#END_EDIT_BLOCK END_ALGORITHM

ALGORITHM aAddAt

VAR_INPUT
 Element : tsElementXY;
 iPos : DINT;
END_VAR

VAR_TEMP
 i : DINT;
END_VAR

VAR
 iStart : DINT;
 iEnd : DINT;
END_VAR
#BEGIN_EDIT_BLOCK
IF NOT mbInit THEN RETURN; END_IF;

IF miNextFree <= miHighBound THEN
    IF iPos < miHighBound AND iPos >= miLowBound THEN

        IF iPos < miNextFree THEN

            iStart := miNextFree;
            iEnd := iPos+1;
        ELSE
            i := iPos;
            iEnd := miNextFree;
        END_IF;
        miNextFree := i + 1;

        //reorganize list
        FOR i := iStart TO iEnd BY -1 DO
            mListStruct.List[i] := mListStruct.List[i-1];
            mListStruct.Used[i] := TRUE;
        END_FOR;
        //adding Element
        mListStruct.List[iPos] := Element;
        mListStruct.Used[iPos] := TRUE;
    ELSE
        //error: out of bounds
        IF sv_TraceLevel.bApplication THEN
            fbDebugTrace(sText := 'ABList.aAddAt: Error: Out of ListBounds');
        END_IF;
    END_IF;
ELSE
    //error: List Full
    SET_ALARM(Name := erListOverflow,
            SubID1 := sv_DeviceId.CompId,
            SubID2 := sv_DeviceId.IndexId,
            Param1 := 'ABList.aAddAt');
END_IF;

;#END_EDIT_BLOCK END_ALGORITHM

ALGORITHM aSearch

VAR_INPUT
 SearchData : tsSearchDataXY;
END_VAR

VAR_OUTPUT
 Element : tsElementXY;
 iPos : DINT;
 bFound : BOOL;
END_VAR

VAR_TEMP
 i : DINT;
END_VAR
#BEGIN_EDIT_BLOCK
IF NOT mbInit THEN RETURN;; END_IF;

iPos := 0;
bFound := FALSE;

FOR i := miLowBound TO miNextFree-1 DO

    IF mListStruct.List[i].SearchData = SearchData THEN

       Element := mListStruct.List[i];
       //remember foundposition for aSearchNext
       miLastFound := i;
       iPos := i;
       bFound := TRUE;
       RETURN;;
    END_IF;
END_FOR;

;#END_EDIT_BLOCK END_ALGORITHM

ALGORITHM aSearchNext

VAR_INPUT
 SearchData : tsSearchDataXY;
END_VAR

VAR_OUTPUT
 Element : tsElementXY;
 iPos : DINT;
 bFound : BOOL;
END_VAR

VAR_TEMP
 i : DINT;
END_VAR
#BEGIN_EDIT_BLOCK
IF NOT mbInit THEN RETURN;; END_IF;

iPos := 0;
bFound := FALSE;

FOR i := miLastFound+1 TO miNextFree-1 DO

    IF mListStruct.List[i].SearchData = SearchData THEN

       Element := mListStruct.List[i];
       //remember foundposition for then next aSearchNext
       miLastFound := i;
       iPos := i;
       bFound := TRUE;
       RETURN;;
    END_IF;
END_FOR;

;#END_EDIT_BLOCK END_ALGORITHM

ALGORITHM aRemove

VAR_INPUT
 SearchData : tsSearchDataXY;
END_VAR

VAR_OUTPUT
 Element : tsElementXY;
 iPos : DINT;
 bFound : BOOL;
END_VAR

VAR_TEMP
 i : DINT;
END_VAR
#BEGIN_EDIT_BLOCK
IF NOT mbInit THEN RETURN; END_IF;

iPos := 0;
bFound := FALSE;

FOR i := miLowBound TO miNextFree-1 DO

    IF mListStruct.List[i].SearchData = SearchData THEN

       iPos := i;
       bFound := TRUE;
       Element := mListStruct.List[i];
       //reorganize list
       FOR i := iPos TO miNextFree-1 DO
           mListStruct.List[i] := mListStruct.List[i+1];
       END_FOR;
       mListStruct.Used[miNextFree-1] := FALSE;
       miNextFree := miNextFree - 1;
       RETURN;
    END_IF;
END_FOR;

;#END_EDIT_BLOCK END_ALGORITHM

ALGORITHM aRemoveAt

VAR_INPUT
 iPos : DINT;
END_VAR

VAR_OUTPUT
 Element : tsElementXY;
END_VAR

VAR_TEMP
 i : DINT;
END_VAR
#BEGIN_EDIT_BLOCK
IF NOT mbInit THEN RETURN; END_IF;

IF iPos <= miHighBound AND iPos >= miLowBound THEN

    Element:= mListStruct.List[iPos];
    miActElement := iPos;

    //reorganize list
    FOR i := iPos TO miNextFree-1 DO
        mListStruct.List[i] := mListStruct.List[i+1];
    END_FOR;
    mListStruct.Used[miNextFree-1] := FALSE;

    miNextFree := miNextFree - 1;
ELSE
    //error: out of bounds
    IF sv_TraceLevel.bApplication THEN
        fbDebugTrace(sText := 'ABList.aRemoveAt: Error: Out of ListBounds');
    END_IF;
END_IF;

;#END_EDIT_BLOCK END_ALGORITHM

ALGORITHM aRemoveAll

VAR_TEMP
 i : DINT;
END_VAR
#BEGIN_EDIT_BLOCK
IF NOT mbInit THEN RETURN; END_IF;
FOR i := miNextFree-1 TO miLowBound DO
    //clearing the whole list
    mListStruct.Used[i] := FALSE;
END_FOR;
miNextFree := miLowBound;

;#END_EDIT_BLOCK END_ALGORITHM

ALGORITHM aElementAt

VAR_OUTPUT
 Element : tsElementXY;
END_VAR

VAR_INPUT
 iPos : DINT;
END_VAR
#BEGIN_EDIT_BLOCK
IF NOT mbInit THEN RETURN; END_IF;

IF iPos <= miHighBound AND iPos >= miLowBound THEN

    Element := mListStruct.List[iPos];
    miActElement := iPos;
ELSE
    //error: out of bounds
    IF sv_TraceLevel.bApplication THEN
        fbDebugTrace(sText := 'ABList.aElementAt: Error: Out of ListBounds');
    END_IF;
END_IF;

;#END_EDIT_BLOCK END_ALGORITHM

ALGORITHM aModifyAt

VAR_INPUT
 iPos : DINT;
END_VAR

VAR_IN_OUT
 Element : tsElementXY;
END_VAR
#BEGIN_EDIT_BLOCK
IF NOT mbInit THEN RETURN; END_IF;

IF iPos <= miHighBound AND iPos >= miLowBound THEN

     mListStruct.List[iPos] := Element;
     miActElement := iPos;
ELSE
    //error: out of bounds
    IF sv_TraceLevel.bApplication THEN
        fbDebugTrace(sText := 'ABList.aModifyAt: Error: Out of ListBounds');
    END_IF;
END_IF;

;#END_EDIT_BLOCK END_ALGORITHM

FUNCTION aGetSize : DINT
 #DUMMY_EDIT_BLOCK
#BEGIN_EDIT_BLOCK
IF NOT mbInit THEN RETURN; END_IF;
//returns the size of the list
aGetSize := miHighBound - miLowBound;

;#END_EDIT_BLOCK END_FUNCTION

FUNCTION aGetElementCount : DINT
 #DUMMY_EDIT_BLOCK
#BEGIN_EDIT_BLOCK
IF NOT mbInit THEN RETURN; END_IF;

aGetElementCount:= miNextFree - miLowBound;

;#END_EDIT_BLOCK END_FUNCTION

ALGORITHM aFirstElement

VAR_OUTPUT
 Element : tsElementXY;
END_VAR
#BEGIN_EDIT_BLOCK
IF NOT mbInit THEN RETURN; END_IF;

miActElement := miLowBound;
Element := mListStruct.List[miLowBound];

;#END_EDIT_BLOCK END_ALGORITHM

ALGORITHM aNextElement

VAR_OUTPUT
 Element : tsElementXY;
 iPos : DINT;
END_VAR
#BEGIN_EDIT_BLOCK
IF NOT mbInit THEN RETURN; END_IF;

IF miActElement < miHighBound THEN

    miActElement := miActElement + 1;
    iPos := miActElement;
    Element := mListStruct.List[miActElement];
END_IF;

;#END_EDIT_BLOCK END_ALGORITHM

ALGORITHM aLastElement

VAR_OUTPUT
 Element : tsElementXY;
END_VAR
#BEGIN_EDIT_BLOCK
IF NOT mbInit THEN RETURN; END_IF;

miActElement := miNextFree - 1;
Element := mListStruct.List[miActElement];

;#END_EDIT_BLOCK END_ALGORITHM

ALGORITHM aPrevElement

VAR_OUTPUT
 Element : tsElementXY;
 iPos : DINT;
END_VAR
#BEGIN_EDIT_BLOCK
IF NOT mbInit THEN RETURN; END_IF;

IF miActElement > miLowBound THEN

    miActElement := miActElement - 1;
    iPos := miActElement;
    Element := mListStruct.List[miActElement];
END_IF;

;#END_EDIT_BLOCK END_ALGORITHM

ALGORITHM aImport

VAR_INPUT
 ListStruct : tsListStructXY;
END_VAR

VAR_TEMP
 i : DINT;
END_VAR
#BEGIN_EDIT_BLOCK
IF NOT mbInit THEN RETURN; END_IF;

miLastFound := miLowBound;
miActElement := miLowBound;
miNextFree := miLowBound;
mListStruct :=  ListStruct;

//cheching used elements
FOR i := miLowBound TO miHighBound DO

   IF NOT mListStruct.Used[i] THEN
        miNextFree := i;
        RETURN;
   END_IF;
END_FOR;

;#END_EDIT_BLOCK END_ALGORITHM

ALGORITHM aExport

VAR_OUTPUT
 ListStruct : tsListStructXY;
END_VAR
#BEGIN_EDIT_BLOCK
IF NOT mbInit THEN RETURN; END_IF;

ListStruct := mListStruct;

;#END_EDIT_BLOCK END_ALGORITHM

END_ALGORITHM_BLOCK

#END_OF_IEC_PART

@Puma @IecEditor 6 10 @Pou 25
@@@BEG_Comment@@@
@h    ! WARNING !
@h    The Kemro K2 system (including software) only meets category B according to EN 954-1,
@h    thus it is not intended for usage in safety-relevant control applications in the field
@h    of personal safety (e.g. emergency stop).
@h    To implement potentially necessary safety-relevant control tasks, always use additional
@h    external safety devices that are intended for the particular purpose, and meet the necessary
@h    functional safety.
@h    For further information see EN 954-1 (EN ISO 13849-1) and/or the K2-x00 user manual, chapter
@h    "CE conformity, directives and standards".

This AB is a model of a list-administration. It provides methods for adding, removing, searching
and fetching listelements.
The list is seperated in 2 dataparts:
- mListStruct.List[x].SearchData
- mListStruct.List[x].ElementData
SearchData is the data which is used for searching an entry in the list.
ElementData is a additional datapart.

The block must be adapted before it is ready for use.
For customizing the list, new listtypes have to be created. (see the models in ListTypes.tu)
This can be done easily by replacing the string "XY" by any list identifier.
Example: To create a Motorlist copy and adapt the datatypes of ListTypes.tu.
          Search and replace "XY" by "Motor"  -> tsListStructMotor.
         Rename ABList.pu and Search and replace "XY" by "Motor".

@@@END_Comment@@@

@BEG_Contents

@BEG_Func
@RT(17)FuncTreeContainer
1
@Var @RT(9)SET_ALARM @RT(0) @T @T @DERIVED 0 @F @RT(23)KEBA_STANDARD_PROCEDURE @F
@T
@BEG_Attrib
0 @RT(0) @RT(0)
@END_Attrib
1 1 @F @F @F @F

@END_Func

@BEG_Const
@RT(18)ConstTreeContainer
0
@END_Const

@BEG_Export

@BEG_Kind
@ALGORITHM_BLOCK @RT(6)ABList @STRUCTURED_TEXT
@RT(0) @RT(0) @RT(0)
@END_Kind

@BEG_Dcl
@RT(16)DclTreeContainer
11
@Var @RT(14)erListOverflow @RT(0) @T @F @DT @RT(5)ALARM @RT(0) @T @T @BASIC 0 @F
@F @F
@T
@BEG_Attrib
3 @RT(0) @RT(0) @RT(0)
@END_Attrib
1 7 @F @F @F @F

@Var @RT(11)mListStruct @RT(0) @T @T @DERIVED 0 @T @T @DT @RT(14)tsListStructXY @RT(0) @T @T @UNKNOWN 0 @F
@F @F
@T
@BEG_Attrib
3 @RT(0) @RT(0) @RT(0)
@END_Attrib
1 0 @F @F @F @F

@Var @RT(10)miNextFree @RT(0) @T @F @DT @RT(4)DINT @RT(0) @T @T @BASIC 0 @F
@F @F
@T
@BEG_Attrib
3 @RT(0) @RT(0) @RT(0)
@END_Attrib
1 0 @F @F @F @F

@Var @RT(10)miLowBound @RT(0) @T @F @DT @RT(4)DINT @RT(0) @T @T @BASIC 0 @F
@F @F
@T
@BEG_Attrib
3 @RT(0) @RT(0) @RT(0)
@END_Attrib
1 0 @F @F @F @F

@Var @RT(11)miHighBound @RT(0) @T @F @DT @RT(4)DINT @RT(0) @T @T @BASIC 0 @F
@F @F
@T
@BEG_Attrib
3 @RT(0) @RT(0) @RT(0)
@END_Attrib
1 0 @F @F @F @F

@Var @RT(6)mbInit @RT(0) @T @F @DT @RT(4)BOOL @RT(0) @T @T @BASIC 0 @F
@F @F
@T
@BEG_Attrib
3 @RT(0) @RT(0) @RT(0)
@END_Attrib
1 0 @F @F @F @F

@Var @RT(11)miLastFound @RT(0) @T @F @DT @RT(4)DINT @RT(0) @T @T @BASIC 0 @F
@F @F
@T
@BEG_Attrib
3 @RT(0) @RT(0) @RT(0)
@END_Attrib
1 0 @F @F @F @F

@Var @RT(12)miActElement @RT(0) @T @F @DT @RT(4)DINT @RT(0) @T @T @BASIC 0 @F
@F @F
@T
@BEG_Attrib
3 @RT(0) @RT(0) @RT(0)
@END_Attrib
1 0 @F @F @F @F

@Var @RT(11)sv_DeviceId @RT(0) @T @T @DERIVED 0 @T @T @DT @RT(10)tsDeviceId @RT(0) @T @T @UNKNOWN 0 @F
@F @F
@T
@BEG_Attrib
3 @RT(0) @RT(0) @RT(0)
@END_Attrib
1 8 @F @F @F @F

@Var @RT(12)fbDebugTrace @RT(0) @T @T @DERIVED 0 @T @T @DT @RT(12)FBDebugTrace @RT(0) @T @T @UNKNOWN 0 @F
@F @F
@T
@BEG_Attrib
3 @RT(0) @RT(0) @RT(0)
@END_Attrib
1 0 @F @F @F @F

@Var @RT(13)sv_TraceLevel @RT(0) @T @T @DERIVED 0 @T @T @DT @RT(12)tsTraceLevel @RT(0) @T @T @UNKNOWN 0 @F
@F @F
@T
@BEG_Attrib
3 @RT(0) @RT(0) @RT(0)
@END_Attrib
1 8 @F @F @F @F

@END_Dcl

@END_Export

@BEG_Body

18

@BEG_Export

@BEG_Algo
@ALGORITHM @RT(5)aInit @STRUCTURED_TEXT
@RT(0) @RT(0) @RT(0) @F @F
@END_Algo

@BEG_Dcl
@RT(16)DclTreeContainer
0
@END_Dcl

@END_Export

@BEG_Export

@BEG_Algo
@ALGORITHM @RT(4)aAdd @STRUCTURED_TEXT
@RT(0) @RT(0) @RT(0) @F @F
@END_Algo

@BEG_Dcl
@RT(16)DclTreeContainer
1
@Var @RT(7)Element @RT(0) @T @T @DERIVED 0 @T @T @DT @RT(11)tsElementXY @RT(0) @T @T @UNKNOWN 0 @F
@F @F
@T
@BEG_Attrib
3 @RT(0) @RT(0) @RT(0)
@END_Attrib
1 1 @F @F @F @F

@END_Dcl

@END_Export

@BEG_Export

@BEG_Algo
@ALGORITHM @RT(6)aAddAt @STRUCTURED_TEXT
@RT(0) @RT(0) @RT(0) @F @F
@END_Algo

@BEG_Dcl
@RT(16)DclTreeContainer
5
@Var @RT(7)Element @RT(0) @T @T @DERIVED 0 @T @T @DT @RT(11)tsElementXY @RT(0) @T @T @UNKNOWN 0 @F
@F @F
@T
@BEG_Attrib
3 @RT(0) @RT(0) @RT(0)
@END_Attrib
1 1 @F @F @F @F

@Var @RT(4)iPos @RT(0) @T @F @DT @RT(4)DINT @RT(0) @T @T @BASIC 0 @F
@F @F
@T
@BEG_Attrib
3 @RT(0) @RT(0) @RT(0)
@END_Attrib
1 1 @F @F @F @F

@Var @RT(1)i @RT(0) @T @F @DT @RT(4)DINT @RT(0) @T @T @BASIC 0 @F
@F @F
@T
@BEG_Attrib
3 @RT(0) @RT(0) @RT(0)
@END_Attrib
1 4 @F @F @F @F

@Var @RT(6)iStart @RT(0) @T @F @DT @RT(4)DINT @RT(0) @T @T @BASIC 0 @F
@F @F
@T
@BEG_Attrib
3 @RT(0) @RT(0) @RT(0)
@END_Attrib
1 0 @F @F @F @F

@Var @RT(4)iEnd @RT(0) @T @F @DT @RT(4)DINT @RT(0) @T @T @BASIC 0 @F
@F @F
@T
@BEG_Attrib
3 @RT(0) @RT(0) @RT(0)
@END_Attrib
1 0 @F @F @F @F

@END_Dcl

@END_Export

@BEG_Export

@BEG_Algo
@ALGORITHM @RT(7)aSearch @STRUCTURED_TEXT
@RT(0) @RT(0) @RT(0) @F @F
@END_Algo

@BEG_Dcl
@RT(16)DclTreeContainer
5
@Var @RT(10)SearchData @RT(0) @T @T @DERIVED 0 @T @T @DT @RT(14)tsSearchDataXY @RT(0) @T @T @UNKNOWN 0 @F
@F @F
@T
@BEG_Attrib
3 @RT(0) @RT(0) @RT(0)
@END_Attrib
1 1 @F @F @F @F

@Var @RT(7)Element @RT(0) @T @T @DERIVED 0 @T @T @DT @RT(11)tsElementXY @RT(0) @T @T @UNKNOWN 0 @F
@F @F
@T
@BEG_Attrib
3 @RT(0) @RT(0) @RT(0)
@END_Attrib
1 3 @F @F @F @F

@Var @RT(4)iPos @RT(0) @T @F @DT @RT(4)DINT @RT(0) @T @T @BASIC 0 @F
@F @F
@T
@BEG_Attrib
3 @RT(0) @RT(0) @RT(0)
@END_Attrib
1 3 @F @F @F @F

@Var @RT(6)bFound @RT(0) @T @F @DT @RT(4)BOOL @RT(0) @T @T @BASIC 0 @F
@F @F
@T
@BEG_Attrib
3 @RT(0) @RT(0) @RT(0)
@END_Attrib
1 3 @F @F @F @F

@Var @RT(1)i @RT(0) @T @F @DT @RT(4)DINT @RT(0) @T @T @BASIC 0 @F
@F @F
@T
@BEG_Attrib
3 @RT(0) @RT(0) @RT(0)
@END_Attrib
1 4 @F @F @F @F

@END_Dcl

@END_Export

@BEG_Export

@BEG_Algo
@ALGORITHM @RT(11)aSearchNext @STRUCTURED_TEXT
@RT(0) @RT(0) @RT(0) @F @F
@END_Algo

@BEG_Dcl
@RT(16)DclTreeContainer
5
@Var @RT(10)SearchData @RT(0) @T @T @DERIVED 0 @T @T @DT @RT(14)tsSearchDataXY @RT(0) @T @T @UNKNOWN 0 @F
@F @F
@T
@BEG_Attrib
3 @RT(0) @RT(0) @RT(0)
@END_Attrib
1 1 @F @F @F @F

@Var @RT(7)Element @RT(0) @T @T @DERIVED 0 @T @T @DT @RT(11)tsElementXY @RT(0) @T @T @UNKNOWN 0 @F
@F @F
@T
@BEG_Attrib
3 @RT(0) @RT(0) @RT(0)
@END_Attrib
1 3 @F @F @F @F

@Var @RT(4)iPos @RT(0) @T @F @DT @RT(4)DINT @RT(0) @T @T @BASIC 0 @F
@F @F
@T
@BEG_Attrib
3 @RT(0) @RT(0) @RT(0)
@END_Attrib
1 3 @F @F @F @F

@Var @RT(6)bFound @RT(0) @T @F @DT @RT(4)BOOL @RT(0) @T @T @BASIC 0 @F
@F @F
@T
@BEG_Attrib
3 @RT(0) @RT(0) @RT(0)
@END_Attrib
1 3 @F @F @F @F

@Var @RT(1)i @RT(0) @T @F @DT @RT(4)DINT @RT(0) @T @T @BASIC 0 @F
@F @F
@T
@BEG_Attrib
3 @RT(0) @RT(0) @RT(0)
@END_Attrib
1 4 @F @F @F @F

@END_Dcl

@END_Export

@BEG_Export

@BEG_Algo
@ALGORITHM @RT(7)aRemove @STRUCTURED_TEXT
@RT(0) @RT(0) @RT(0) @F @F
@END_Algo

@BEG_Dcl
@RT(16)DclTreeContainer
5
@Var @RT(10)SearchData @RT(0) @T @T @DERIVED 0 @T @T @DT @RT(14)tsSearchDataXY @RT(0) @T @T @UNKNOWN 0 @F
@F @F
@T
@BEG_Attrib
3 @RT(0) @RT(0) @RT(0)
@END_Attrib
1 1 @F @F @F @F

@Var @RT(7)Element @RT(0) @T @T @DERIVED 0 @T @T @DT @RT(11)tsElementXY @RT(0) @T @T @UNKNOWN 0 @F
@F @F
@T
@BEG_Attrib
3 @RT(0) @RT(0) @RT(0)
@END_Attrib
1 3 @F @F @F @F

@Var @RT(4)iPos @RT(0) @T @F @DT @RT(4)DINT @RT(0) @T @T @BASIC 0 @F
@F @F
@T
@BEG_Attrib
3 @RT(0) @RT(0) @RT(0)
@END_Attrib
1 3 @F @F @F @F

@Var @RT(6)bFound @RT(0) @T @F @DT @RT(4)BOOL @RT(0) @T @T @BASIC 0 @F
@F @F
@T
@BEG_Attrib
3 @RT(0) @RT(0) @RT(0)
@END_Attrib
1 3 @F @F @F @F

@Var @RT(1)i @RT(0) @T @F @DT @RT(4)DINT @RT(0) @T @T @BASIC 0 @F
@F @F
@T
@BEG_Attrib
3 @RT(0) @RT(0) @RT(0)
@END_Attrib
1 4 @F @F @F @F

@END_Dcl

@END_Export

@BEG_Export

@BEG_Algo
@ALGORITHM @RT(9)aRemoveAt @STRUCTURED_TEXT
@RT(0) @RT(0) @RT(0) @F @F
@END_Algo

@BEG_Dcl
@RT(16)DclTreeContainer
3
@Var @RT(4)iPos @RT(0) @T @F @DT @RT(4)DINT @RT(0) @T @T @BASIC 0 @F
@F @F
@T
@BEG_Attrib
3 @RT(0) @RT(0) @RT(0)
@END_Attrib
1 1 @F @F @F @F

@Var @RT(7)Element @RT(0) @T @T @DERIVED 0 @T @T @DT @RT(11)tsElementXY @RT(0) @T @T @UNKNOWN 0 @F
@F @F
@T
@BEG_Attrib
3 @RT(0) @RT(0) @RT(0)
@END_Attrib
1 3 @F @F @F @F

@Var @RT(1)i @RT(0) @T @F @DT @RT(4)DINT @RT(0) @T @T @BASIC 0 @F
@F @F
@T
@BEG_Attrib
3 @RT(0) @RT(0) @RT(0)
@END_Attrib
1 4 @F @F @F @F

@END_Dcl

@END_Export

@BEG_Export

@BEG_Algo
@ALGORITHM @RT(10)aRemoveAll @STRUCTURED_TEXT
@RT(0) @RT(0) @RT(0) @F @F
@END_Algo

@BEG_Dcl
@RT(16)DclTreeContainer
1
@Var @RT(1)i @RT(0) @T @F @DT @RT(4)DINT @RT(0) @T @T @BASIC 0 @F
@F @F
@T
@BEG_Attrib
3 @RT(0) @RT(0) @RT(0)
@END_Attrib
1 4 @F @F @F @F

@END_Dcl

@END_Export

@BEG_Export

@BEG_Algo
@ALGORITHM @RT(10)aElementAt @STRUCTURED_TEXT
@RT(0) @RT(0) @RT(0) @F @F
@END_Algo

@BEG_Dcl
@RT(16)DclTreeContainer
2
@Var @RT(7)Element @RT(0) @T @T @DERIVED 0 @T @T @DT @RT(11)tsElementXY @RT(0) @T @T @UNKNOWN 0 @F
@F @F
@T
@BEG_Attrib
3 @RT(0) @RT(0) @RT(0)
@END_Attrib
1 3 @F @F @F @F

@Var @RT(4)iPos @RT(0) @T @F @DT @RT(4)DINT @RT(0) @T @T @BASIC 0 @F
@F @F
@T
@BEG_Attrib
3 @RT(0) @RT(0) @RT(0)
@END_Attrib
1 1 @F @F @F @F

@END_Dcl

@END_Export

@BEG_Export

@BEG_Algo
@ALGORITHM @RT(9)aModifyAt @STRUCTURED_TEXT
@RT(0) @RT(0) @RT(0) @F @F
@END_Algo

@BEG_Dcl
@RT(16)DclTreeContainer
2
@Var @RT(4)iPos @RT(0) @T @F @DT @RT(4)DINT @RT(0) @T @T @BASIC 0 @F
@F @F
@T
@BEG_Attrib
3 @RT(0) @RT(0) @RT(0)
@END_Attrib
1 1 @F @F @F @F

@Var @RT(7)Element @RT(0) @T @T @DERIVED 0 @T @T @DT @RT(11)tsElementXY @RT(0) @T @T @UNKNOWN 0 @F
@F @F
@T
@BEG_Attrib
3 @RT(0) @RT(0) @RT(0)
@END_Attrib
1 2 @F @F @F @F

@END_Dcl

@END_Export

@BEG_Export

@BEG_Algo
@FUNCTION @RT(8)aGetSize @STRUCTURED_TEXT
@RT(4)DINT @RT(0) @RT(0) @F @F
@END_Algo

@BEG_Dcl
@RT(16)DclTreeContainer
0
@END_Dcl

@END_Export

@BEG_Export

@BEG_Algo
@FUNCTION @RT(16)aGetElementCount @STRUCTURED_TEXT
@RT(4)DINT @RT(0) @RT(0) @F @F
@END_Algo

@BEG_Dcl
@RT(16)DclTreeContainer
0
@END_Dcl

@END_Export

@BEG_Export

@BEG_Algo
@ALGORITHM @RT(13)aFirstElement @STRUCTURED_TEXT
@RT(0) @RT(0) @RT(0) @F @F
@END_Algo

@BEG_Dcl
@RT(16)DclTreeContainer
1
@Var @RT(7)Element @RT(0) @T @T @DERIVED 0 @T @T @DT @RT(11)tsElementXY @RT(0) @T @T @UNKNOWN 0 @F
@F @F
@T
@BEG_Attrib
3 @RT(0) @RT(0) @RT(0)
@END_Attrib
1 3 @F @F @F @F

@END_Dcl

@END_Export

@BEG_Export

@BEG_Algo
@ALGORITHM @RT(12)aNextElement @STRUCTURED_TEXT
@RT(0) @RT(0) @RT(0) @F @F
@END_Algo

@BEG_Dcl
@RT(16)DclTreeContainer
2
@Var @RT(7)Element @RT(0) @T @T @DERIVED 0 @T @T @DT @RT(11)tsElementXY @RT(0) @T @T @UNKNOWN 0 @F
@F @F
@T
@BEG_Attrib
3 @RT(0) @RT(0) @RT(0)
@END_Attrib
1 3 @F @F @F @F

@Var @RT(4)iPos @RT(0) @T @F @DT @RT(4)DINT @RT(0) @T @T @BASIC 0 @F
@F @F
@T
@BEG_Attrib
3 @RT(0) @RT(0) @RT(0)
@END_Attrib
1 3 @F @F @F @F

@END_Dcl

@END_Export

@BEG_Export

@BEG_Algo
@ALGORITHM @RT(12)aLastElement @STRUCTURED_TEXT
@RT(0) @RT(0) @RT(0) @F @F
@END_Algo

@BEG_Dcl
@RT(16)DclTreeContainer
1
@Var @RT(7)Element @RT(0) @T @T @DERIVED 0 @T @T @DT @RT(11)tsElementXY @RT(0) @T @T @UNKNOWN 0 @F
@F @F
@T
@BEG_Attrib
3 @RT(0) @RT(0) @RT(0)
@END_Attrib
1 3 @F @F @F @F

@END_Dcl

@END_Export

@BEG_Export

@BEG_Algo
@ALGORITHM @RT(12)aPrevElement @STRUCTURED_TEXT
@RT(0) @RT(0) @RT(0) @F @F
@END_Algo

@BEG_Dcl
@RT(16)DclTreeContainer
2
@Var @RT(7)Element @RT(0) @T @T @DERIVED 0 @T @T @DT @RT(11)tsElementXY @RT(0) @T @T @UNKNOWN 0 @F
@F @F
@T
@BEG_Attrib
3 @RT(0) @RT(0) @RT(0)
@END_Attrib
1 3 @F @F @F @F

@Var @RT(4)iPos @RT(0) @T @F @DT @RT(4)DINT @RT(0) @T @T @BASIC 0 @F
@F @F
@T
@BEG_Attrib
3 @RT(0) @RT(0) @RT(0)
@END_Attrib
1 3 @F @F @F @F

@END_Dcl

@END_Export

@BEG_Export

@BEG_Algo
@ALGORITHM @RT(7)aImport @STRUCTURED_TEXT
@RT(0) @RT(0) @RT(0) @F @F
@END_Algo

@BEG_Dcl
@RT(16)DclTreeContainer
2
@Var @RT(10)ListStruct @RT(0) @T @T @DERIVED 0 @T @T @DT @RT(14)tsListStructXY @RT(0) @T @T @UNKNOWN 0 @F
@F @F
@T
@BEG_Attrib
3 @RT(0) @RT(0) @RT(0)
@END_Attrib
1 1 @F @F @F @F

@Var @RT(1)i @RT(0) @T @F @DT @RT(4)DINT @RT(0) @T @T @BASIC 0 @F
@F @F
@T
@BEG_Attrib
3 @RT(0) @RT(0) @RT(0)
@END_Attrib
1 4 @F @F @F @F

@END_Dcl

@END_Export

@BEG_Export

@BEG_Algo
@ALGORITHM @RT(7)aExport @STRUCTURED_TEXT
@RT(0) @RT(0) @RT(0) @F @F
@END_Algo

@BEG_Dcl
@RT(16)DclTreeContainer
1
@Var @RT(10)ListStruct @RT(0) @T @T @DERIVED 0 @T @T @DT @RT(14)tsListStructXY @RT(0) @T @T @UNKNOWN 0 @F
@F @F
@T
@BEG_Attrib
3 @RT(0) @RT(0) @RT(0)
@END_Attrib
1 3 @F @F @F @F

@END_Dcl

@END_Export

@BEG_Body
@TL(7)
miLowBound := GET_LOW_BOUND(mListStruct.List);
miHighBound := GET_HIGH_BOUND(mListStruct.List);
miNextFree := miLowBound;
miLastFound := miLowBound;
miActElement := miLowBound;
mbInit := TRUE;

@END_Body

@@@BEG_Comment@@@
@TL(0)

@@@END_Comment@@@

@BEG_Body
@TL(15)
IF NOT mbInit THEN RETURN;; END_IF;

IF miNextFree < miHighBound THEN

    mListStruct.List[miNextFree] := Element;
    mListStruct.Used[miNextFree] := TRUE;
    miNextFree := miNextFree + 1;
ELSE
    //error: List Full
    SET_ALARM(Name := erListOverflow,
              SubID1 := sv_DeviceId.CompId,
              SubID2 := sv_DeviceId.IndexId,
              Param1 := 'ABList.aAdd');
END_IF;

@END_Body

@@@BEG_Comment@@@
@TL(0)

@@@END_Comment@@@

@BEG_Body
@TL(37)
IF NOT mbInit THEN RETURN; END_IF;

IF miNextFree <= miHighBound THEN
    IF iPos < miHighBound AND iPos >= miLowBound THEN

        IF iPos < miNextFree THEN

            iStart := miNextFree;
            iEnd := iPos+1;
        ELSE
            i := iPos;
            iEnd := miNextFree;
        END_IF;
        miNextFree := i + 1;

        //reorganize list
        FOR i := iStart TO iEnd BY -1 DO
            mListStruct.List[i] := mListStruct.List[i-1];
            mListStruct.Used[i] := TRUE;
        END_FOR;
        //adding Element
        mListStruct.List[iPos] := Element;
        mListStruct.Used[iPos] := TRUE;
    ELSE
        //error: out of bounds
        IF sv_TraceLevel.bApplication THEN
            fbDebugTrace(sText := 'ABList.aAddAt: Error: Out of ListBounds');
        END_IF;
    END_IF;
ELSE
    //error: List Full
    SET_ALARM(Name := erListOverflow,
            SubID1 := sv_DeviceId.CompId,
            SubID2 := sv_DeviceId.IndexId,
            Param1 := 'ABList.aAddAt');
END_IF;

@END_Body

@@@BEG_Comment@@@
@TL(0)

@@@END_Comment@@@

@BEG_Body
@TL(18)
IF NOT mbInit THEN RETURN;; END_IF;

iPos := 0;
bFound := FALSE;

FOR i := miLowBound TO miNextFree-1 DO

    IF mListStruct.List[i].SearchData = SearchData THEN

       Element := mListStruct.List[i];
       //remember foundposition for aSearchNext
       miLastFound := i;
       iPos := i;
       bFound := TRUE;
       RETURN;;
    END_IF;
END_FOR;

@END_Body

@@@BEG_Comment@@@
@TL(0)

@@@END_Comment@@@

@BEG_Body
@TL(19)
IF NOT mbInit THEN RETURN;; END_IF;

iPos := 0;
bFound := FALSE;

FOR i := miLastFound+1 TO miNextFree-1 DO

    IF mListStruct.List[i].SearchData = SearchData THEN

       Element := mListStruct.List[i];
       //remember foundposition for then next aSearchNext
       miLastFound := i;
       iPos := i;
       bFound := TRUE;
       RETURN;;
    END_IF;
END_FOR;

@END_Body

@@@BEG_Comment@@@
@TL(0)

@@@END_Comment@@@

@BEG_Body
@TL(22)
IF NOT mbInit THEN RETURN; END_IF;

iPos := 0;
bFound := FALSE;

FOR i := miLowBound TO miNextFree-1 DO

    IF mListStruct.List[i].SearchData = SearchData THEN

       iPos := i;
       bFound := TRUE;
       Element := mListStruct.List[i];
       //reorganize list
       FOR i := iPos TO miNextFree-1 DO
           mListStruct.List[i] := mListStruct.List[i+1];
       END_FOR;
       mListStruct.Used[miNextFree-1] := FALSE;
       miNextFree := miNextFree - 1;
       RETURN;
    END_IF;
END_FOR;

@END_Body

@@@BEG_Comment@@@
@TL(0)

@@@END_Comment@@@

@BEG_Body
@TL(21)
IF NOT mbInit THEN RETURN; END_IF;

IF iPos <= miHighBound AND iPos >= miLowBound THEN

    Element:= mListStruct.List[iPos];
    miActElement := iPos;

    //reorganize list
    FOR i := iPos TO miNextFree-1 DO
        mListStruct.List[i] := mListStruct.List[i+1];
    END_FOR;
    mListStruct.Used[miNextFree-1] := FALSE;

    miNextFree := miNextFree - 1;
ELSE
    //error: out of bounds
    IF sv_TraceLevel.bApplication THEN
        fbDebugTrace(sText := 'ABList.aRemoveAt: Error: Out of ListBounds');
    END_IF;
END_IF;

@END_Body

@@@BEG_Comment@@@
@TL(0)

@@@END_Comment@@@

@BEG_Body
@TL(7)
IF NOT mbInit THEN RETURN; END_IF;
FOR i := miNextFree-1 TO miLowBound DO
    //clearing the whole list
    mListStruct.Used[i] := FALSE;
END_FOR;
miNextFree := miLowBound;

@END_Body

@@@BEG_Comment@@@
@TL(0)

@@@END_Comment@@@

@BEG_Body
@TL(13)
IF NOT mbInit THEN RETURN; END_IF;

IF iPos <= miHighBound AND iPos >= miLowBound THEN

    Element := mListStruct.List[iPos];
    miActElement := iPos;
ELSE
    //error: out of bounds
    IF sv_TraceLevel.bApplication THEN
        fbDebugTrace(sText := 'ABList.aElementAt: Error: Out of ListBounds');
    END_IF;
END_IF;

@END_Body

@@@BEG_Comment@@@
@TL(0)

@@@END_Comment@@@

@BEG_Body
@TL(13)
IF NOT mbInit THEN RETURN; END_IF;

IF iPos <= miHighBound AND iPos >= miLowBound THEN

     mListStruct.List[iPos] := Element;
     miActElement := iPos;
ELSE
    //error: out of bounds
    IF sv_TraceLevel.bApplication THEN
        fbDebugTrace(sText := 'ABList.aModifyAt: Error: Out of ListBounds');
    END_IF;
END_IF;

@END_Body

@@@BEG_Comment@@@
@TL(0)

@@@END_Comment@@@

@BEG_Body
@TL(5)
IF NOT mbInit THEN RETURN; END_IF;
//returns the size of the list
aGetSize := miHighBound - miLowBound;

@END_Body

@@@BEG_Comment@@@
@TL(0)

@@@END_Comment@@@

@BEG_Body
@TL(5)
IF NOT mbInit THEN RETURN; END_IF;

aGetElementCount:= miNextFree - miLowBound;

@END_Body

@@@BEG_Comment@@@
@TL(0)

@@@END_Comment@@@

@BEG_Body
@TL(6)
IF NOT mbInit THEN RETURN; END_IF;

miActElement := miLowBound;
Element := mListStruct.List[miLowBound];

@END_Body

@@@BEG_Comment@@@
@TL(0)

@@@END_Comment@@@

@BEG_Body
@TL(9)
IF NOT mbInit THEN RETURN; END_IF;

IF miActElement < miHighBound THEN

    miActElement := miActElement + 1;
    iPos := miActElement;
    Element := mListStruct.List[miActElement];
END_IF;

@END_Body

@@@BEG_Comment@@@
@TL(0)

@@@END_Comment@@@

@BEG_Body
@TL(6)
IF NOT mbInit THEN RETURN; END_IF;

miActElement := miNextFree - 1;
Element := mListStruct.List[miActElement];

@END_Body

@@@BEG_Comment@@@
@TL(0)

@@@END_Comment@@@

@BEG_Body
@TL(9)
IF NOT mbInit THEN RETURN; END_IF;

IF miActElement > miLowBound THEN

    miActElement := miActElement - 1;
    iPos := miActElement;
    Element := mListStruct.List[miActElement];
END_IF;

@END_Body

@@@BEG_Comment@@@
@TL(0)

@@@END_Comment@@@

@BEG_Body
@TL(16)
IF NOT mbInit THEN RETURN; END_IF;

miLastFound := miLowBound;
miActElement := miLowBound;
miNextFree := miLowBound;
mListStruct :=  ListStruct;

//cheching used elements
FOR i := miLowBound TO miHighBound DO

   IF NOT mListStruct.Used[i] THEN
        miNextFree := i;
        RETURN;
   END_IF;
END_FOR;

@END_Body

@@@BEG_Comment@@@
@TL(0)

@@@END_Comment@@@

@BEG_Body
@TL(4)
IF NOT mbInit THEN RETURN; END_IF;

ListStruct := mListStruct;

@END_Body

@@@BEG_Comment@@@
@TL(0)

@@@END_Comment@@@
@END_Body

@END_Contents
